{attribute addProperty BoxType "EK1100-0000-0018"}
{attribute addProperty Id "Beckhoff_EL34xxEK1122Beckhoff_EL34xxEK1122_54E02F3C162A_0001_EL3403_0000_0017EL3403_4661793D60275.25A_0002_EL3403_0000_0018EL3403_602DA43960275.25A_0003_EL3403_0000_0019EL3403_602DA43960275.25A_0004_EL3403_0000_0020EL3403_602DA43960275.25A_0005_EL3403_0000_0021EL3403_602DA43960275.25A_0006_EL3403_0000_0022EL3403_6F016EBB57071.25A_0007_EL3403_0000_0023EL3403_6F016EBB57071.25A_0008_EL3403_0010_0017EL3403_4661793D60275.25A_0009_EL3403_0010_0018EL3403_602DA43960275.25A_0010_EL3403_0010_0019EL3403_602DA43960275.25A_0011_EL3403_0010_0020EL3403_602DA43960275.25A_0012_EL3403_0010_0021EL3403_602DA43960275.25A_0013_EL3403_0010_0022EL3403_6F016EBB57071.25A_0014_EL3403_0010_0023EL3403_6F016EBB57071.25A_0015_EL3403_0010_0024EL3403_6F016EBB57071.25A_0016_EL3403_0026_0017EL3403_4661793D60275.25A_0017_EL3403_0026_0018EL3403_602DA43960275.25A_0018_EL3403_0026_0019EL3403_602DA43960275.25A_0019_EL3403_0026_0020EL3403_602DA43960275.25A_0020_EL3403_0026_0021EL3403_602DA43960275.25A_0021_EL3403_0026_0022EL3403_6F016EBB57071.25A_0022_EL3403_0026_0023EL3403_6F016EBB57071.25A_0023_EL3403_0026_0024EL3403_6F016EBB57071.25A_0024_EL3403_0100_0017EL3403_4661793D60275.25A_0025_EL3403_0100_0018EL3403_602DA43960275.25A_0026_EL3403_0100_0019EL3403_602DA43960275.25A_0027_EL3403_0100_0020EL3403_602DA43960275.25A_0028_EL3403_0100_0021EL3403_602DA43960275.25A_0029_EL3403_0100_0022EL3403_6F016EBB57071.25A_0030_EL3403_0100_0023EL3403_6F016EBB57071.25A_0031_EL3403_0100_0024EL3403_6F016EBB57071.25A_0032_EL3403_0111_0017EL3403_4661793D60275.25A_0033_EL3403_0111_0018EL3403_602DA43960275.25A_0034_EL3403_0111_0019EL3403_602DA43960275.25A_0035_EL3403_0111_0020EL3403_602DA43960275.25A_0036_EL3403_0111_0021EL3403_602DA43960275.25A_0037_EL3403_0111_0022EL3403_6F016EBB57071.25A_0038_EL3403_0111_0023EL3403_6F016EBB57071.25A_0039_EL3403_0111_0024EL3403_6F016EBB57071.25A_0040_EL3403_0126_0017EL3403_4661793D60275.25A_0041_EL3403_0126_0018EL3403_602DA43960275.25A_0042_EL3403_0126_0019EL3403_602DA43960275.25A_0043_EL3403_0126_0020EL3403_602DA43960275.25A_0044_EL3403_0126_0021EL3403_602DA43960275.25A_0045_EL3403_0126_0022EL3403_6F016EBB57071.25A_0046_EL3403_0126_0023EL3403_6F016EBB57071.25A_0047_EL3403_0126_0024EL3403_6F016EBB57071.25A_0048_EL3403_0333_0023EL3403_6F016EBB57071.25A_0049_EL3403_0333_0024EL3403_6F016EBB57071.25A_0050_EL3413_0000_0016EL3413_DFA511C864280.25A_0051_EL3413_0000_0017EL3413_DFA511C864280.25A_0052_EL3413_0000_0018EL3413_DFA511C864280.25A_0053_EL3413_0000_0019EL3413_BFE9962F64280.25A_0054_EL3413_0000_0020EL3413_BFE9962F64280.25A_0055_EL3413_0001_0016EL3413_BFE9962F64280.25A_0056_EL3413_0001_0017EL3413_BFE9962F64280.25A_0057_EL3413_0120_0017EL3413_DFA511C864280.25A_0058_EL3413_0001_0018EL3413_BFE9962F64280.25A_0059_EL3413_0120_0018EL3413_BFE9962F64280.25A_0060_EL3413_0120_0019EL3413_BFE9962F64280.25A_0061_EL3423_0000_0016EL3423_8712F12C1506188.25A_0062_EL3423_0000_0017EL3423_C8A9BC881506188.25A_0063_EL3423_0000_0018EL3423_C8A9BC881506188.25A_0064_EL3423_0000_0019EL3423_C8A9BC881506188.25A_0065_EL3423_0000_0020EL3423_AE18C60F930116.25A_0066_EL3423_0000_0021EL3423_AE18C60F930116.25A_0067_EL3433_0000_0016EL3433_BFE9962F64280.25A_0068_EL3433_0000_0017EL3433_BFE9962F64280.25A_0069_EL3433_0000_0018EL3433_BFE9962F64280.25A_0070_EL3443_0000_0016EL3443_2BD502B51650206.25A_0071_EL3443_0000_0017EL3443_538373741650206.25A_0072_EL3443_0000_0018EL3443_538373741650206.25A_0073_EL3443_0000_0019EL3443_538373741650206.25A_0074_EL3443_0000_0020EL3443_2BD502B51650206.25A_0075_EL3443_0000_0021EL3443_2BD502B51650206.25A_0076_EL3443_0010_0016EL3443_2BD502B51650206.25A_0077_EL3443_0010_0017EL3443_538373741650206.25A_0078_EL3443_0010_0018EL3443_538373741650206.25A_0079_EL3443_0010_0019EL3443_538373741650206.25A_0080_EL3443_0010_0020EL3443_2BD502B51650206.25A_0081_EL3443_0010_0021EL3443_2BD502B51650206.25A_0082_EL3443_0011_0018EL3443_538373741650206.25A_0083_EL3443_0011_0019EL3443_538373741650206.25A_0084_EL3443_0011_0020EL3443_2BD502B51650206.25A_0085_EL3443_0011_0021EL3443_2BD502B51650206.25A_0086_EL3443_0013_0018EL3443_538373741650206.25A_0087_EL3443_0013_0019EL3443_538373741650206.25A_0088_EL3443_0013_0020EL3443_2BD502B51650206.25A_0089_EL3443_0013_0021EL3443_2BD502B51650206.25A_0090_EL3446_0000_0016EL3446_80BBA9A057872.25A_0091_EL3446_0000_0017EL3446_80BBA9A057872.25A_0092_EL3453_0000_0017EL3453_10B71D421202150.25A_0093_EL3453_0000_0018EL3453_BDDFEB0B1194149.25A_0094_EL3453_0000_0019EL3453_BDDFEB0B1194149.25A_0095_EL3453_0000_0020EL3453_10B71D421202150.25A_0096_EL3453_0000_0021EL3453_10B71D421202150.25A_0097_EL3453_0100_0021EL3453_10B71D421202150.25A_0098_EL3483_0000_0016EL3483_4A23656431439.25A_0099_EL3483_0000_0017EL3483_4A23656431439.25A_0100_EL3483_0000_0018EL3483_4A23656431439.25A_0101_EL3483_0000_0019EL3483_4A23656431439.25A_0102_EL3483_0000_0020EL3483_4A23656431439.25A_0103_EL3483_0000_0021EL3483_4A23656431439.25A_0104_EL3483_0060_0018EL3483_2724D36850663.25A_0105_EL3483_0060_0019EL3483_2724D36850663.25A_0106_EL3483_0060_0020EL3483_EF2C452150663.25A_0107_EL3483_0060_0021EL3483_EF2C452150663.25"}
{attribute addProperty CRC "1278133200"}
{attribute addProperty SizeInBites "91038"}
{attribute addProperty SizeInBytes "11379.75"}
TYPE Beckhoff_EL34xx_4C2EC3D0 EXTENDS EK1100_179A0949 :
STRUCT
	{attribute addProperty Name "Beckhoff_EL34xxEK1122"}
	Beckhoff_EL34xxEK1122 : Beckhoff_EL34xxEK1122_54E02F3C;
	{attribute addProperty Name "A_0001_EL3403_0000_0017"}
	A_0001_EL3403_0000_0017 : EL3403_4661793D;
	{attribute addProperty Name "A_0002_EL3403_0000_0018"}
	A_0002_EL3403_0000_0018 : EL3403_602DA439;
	{attribute addProperty Name "A_0003_EL3403_0000_0019"}
	A_0003_EL3403_0000_0019 : EL3403_602DA439;
	{attribute addProperty Name "A_0004_EL3403_0000_0020"}
	A_0004_EL3403_0000_0020 : EL3403_602DA439;
	{attribute addProperty Name "A_0005_EL3403_0000_0021"}
	A_0005_EL3403_0000_0021 : EL3403_602DA439;
	{attribute addProperty Name "A_0006_EL3403_0000_0022"}
	A_0006_EL3403_0000_0022 : EL3403_6F016EBB;
	{attribute addProperty Name "A_0007_EL3403_0000_0023"}
	A_0007_EL3403_0000_0023 : EL3403_6F016EBB;
	{attribute addProperty Name "A_0008_EL3403_0010_0017"}
	A_0008_EL3403_0010_0017 : EL3403_4661793D;
	{attribute addProperty Name "A_0009_EL3403_0010_0018"}
	A_0009_EL3403_0010_0018 : EL3403_602DA439;
	{attribute addProperty Name "A_0010_EL3403_0010_0019"}
	A_0010_EL3403_0010_0019 : EL3403_602DA439;
	{attribute addProperty Name "A_0011_EL3403_0010_0020"}
	A_0011_EL3403_0010_0020 : EL3403_602DA439;
	{attribute addProperty Name "A_0012_EL3403_0010_0021"}
	A_0012_EL3403_0010_0021 : EL3403_602DA439;
	{attribute addProperty Name "A_0013_EL3403_0010_0022"}
	A_0013_EL3403_0010_0022 : EL3403_6F016EBB;
	{attribute addProperty Name "A_0014_EL3403_0010_0023"}
	A_0014_EL3403_0010_0023 : EL3403_6F016EBB;
	{attribute addProperty Name "A_0015_EL3403_0010_0024"}
	A_0015_EL3403_0010_0024 : EL3403_6F016EBB;
	{attribute addProperty Name "A_0016_EL3403_0026_0017"}
	A_0016_EL3403_0026_0017 : EL3403_4661793D;
	{attribute addProperty Name "A_0017_EL3403_0026_0018"}
	A_0017_EL3403_0026_0018 : EL3403_602DA439;
	{attribute addProperty Name "A_0018_EL3403_0026_0019"}
	A_0018_EL3403_0026_0019 : EL3403_602DA439;
	{attribute addProperty Name "A_0019_EL3403_0026_0020"}
	A_0019_EL3403_0026_0020 : EL3403_602DA439;
	{attribute addProperty Name "A_0020_EL3403_0026_0021"}
	A_0020_EL3403_0026_0021 : EL3403_602DA439;
	{attribute addProperty Name "A_0021_EL3403_0026_0022"}
	A_0021_EL3403_0026_0022 : EL3403_6F016EBB;
	{attribute addProperty Name "A_0022_EL3403_0026_0023"}
	A_0022_EL3403_0026_0023 : EL3403_6F016EBB;
	{attribute addProperty Name "A_0023_EL3403_0026_0024"}
	A_0023_EL3403_0026_0024 : EL3403_6F016EBB;
	{attribute addProperty Name "A_0024_EL3403_0100_0017"}
	A_0024_EL3403_0100_0017 : EL3403_4661793D;
	{attribute addProperty Name "A_0025_EL3403_0100_0018"}
	A_0025_EL3403_0100_0018 : EL3403_602DA439;
	{attribute addProperty Name "A_0026_EL3403_0100_0019"}
	A_0026_EL3403_0100_0019 : EL3403_602DA439;
	{attribute addProperty Name "A_0027_EL3403_0100_0020"}
	A_0027_EL3403_0100_0020 : EL3403_602DA439;
	{attribute addProperty Name "A_0028_EL3403_0100_0021"}
	A_0028_EL3403_0100_0021 : EL3403_602DA439;
	{attribute addProperty Name "A_0029_EL3403_0100_0022"}
	A_0029_EL3403_0100_0022 : EL3403_6F016EBB;
	{attribute addProperty Name "A_0030_EL3403_0100_0023"}
	A_0030_EL3403_0100_0023 : EL3403_6F016EBB;
	{attribute addProperty Name "A_0031_EL3403_0100_0024"}
	A_0031_EL3403_0100_0024 : EL3403_6F016EBB;
	{attribute addProperty Name "A_0032_EL3403_0111_0017"}
	A_0032_EL3403_0111_0017 : EL3403_4661793D;
	{attribute addProperty Name "A_0033_EL3403_0111_0018"}
	A_0033_EL3403_0111_0018 : EL3403_602DA439;
	{attribute addProperty Name "A_0034_EL3403_0111_0019"}
	A_0034_EL3403_0111_0019 : EL3403_602DA439;
	{attribute addProperty Name "A_0035_EL3403_0111_0020"}
	A_0035_EL3403_0111_0020 : EL3403_602DA439;
	{attribute addProperty Name "A_0036_EL3403_0111_0021"}
	A_0036_EL3403_0111_0021 : EL3403_602DA439;
	{attribute addProperty Name "A_0037_EL3403_0111_0022"}
	A_0037_EL3403_0111_0022 : EL3403_6F016EBB;
	{attribute addProperty Name "A_0038_EL3403_0111_0023"}
	A_0038_EL3403_0111_0023 : EL3403_6F016EBB;
	{attribute addProperty Name "A_0039_EL3403_0111_0024"}
	A_0039_EL3403_0111_0024 : EL3403_6F016EBB;
	{attribute addProperty Name "A_0040_EL3403_0126_0017"}
	A_0040_EL3403_0126_0017 : EL3403_4661793D;
	{attribute addProperty Name "A_0041_EL3403_0126_0018"}
	A_0041_EL3403_0126_0018 : EL3403_602DA439;
	{attribute addProperty Name "A_0042_EL3403_0126_0019"}
	A_0042_EL3403_0126_0019 : EL3403_602DA439;
	{attribute addProperty Name "A_0043_EL3403_0126_0020"}
	A_0043_EL3403_0126_0020 : EL3403_602DA439;
	{attribute addProperty Name "A_0044_EL3403_0126_0021"}
	A_0044_EL3403_0126_0021 : EL3403_602DA439;
	{attribute addProperty Name "A_0045_EL3403_0126_0022"}
	A_0045_EL3403_0126_0022 : EL3403_6F016EBB;
	{attribute addProperty Name "A_0046_EL3403_0126_0023"}
	A_0046_EL3403_0126_0023 : EL3403_6F016EBB;
	{attribute addProperty Name "A_0047_EL3403_0126_0024"}
	A_0047_EL3403_0126_0024 : EL3403_6F016EBB;
	{attribute addProperty Name "A_0048_EL3403_0333_0023"}
	A_0048_EL3403_0333_0023 : EL3403_6F016EBB;
	{attribute addProperty Name "A_0049_EL3403_0333_0024"}
	A_0049_EL3403_0333_0024 : EL3403_6F016EBB;
	{attribute addProperty Name "A_0050_EL3413_0000_0016"}
	A_0050_EL3413_0000_0016 : EL3413_DFA511C8;
	{attribute addProperty Name "A_0051_EL3413_0000_0017"}
	A_0051_EL3413_0000_0017 : EL3413_DFA511C8;
	{attribute addProperty Name "A_0052_EL3413_0000_0018"}
	A_0052_EL3413_0000_0018 : EL3413_DFA511C8;
	{attribute addProperty Name "A_0053_EL3413_0000_0019"}
	A_0053_EL3413_0000_0019 : EL3413_BFE9962F;
	{attribute addProperty Name "A_0054_EL3413_0000_0020"}
	A_0054_EL3413_0000_0020 : EL3413_BFE9962F;
	{attribute addProperty Name "A_0055_EL3413_0001_0016"}
	A_0055_EL3413_0001_0016 : EL3413_BFE9962F;
	{attribute addProperty Name "A_0056_EL3413_0001_0017"}
	A_0056_EL3413_0001_0017 : EL3413_BFE9962F;
	{attribute addProperty Name "A_0057_EL3413_0120_0017"}
	A_0057_EL3413_0120_0017 : EL3413_DFA511C8;
	{attribute addProperty Name "A_0058_EL3413_0001_0018"}
	A_0058_EL3413_0001_0018 : EL3413_BFE9962F;
	{attribute addProperty Name "A_0059_EL3413_0120_0018"}
	A_0059_EL3413_0120_0018 : EL3413_BFE9962F;
	{attribute addProperty Name "A_0060_EL3413_0120_0019"}
	A_0060_EL3413_0120_0019 : EL3413_BFE9962F;
	{attribute addProperty Name "A_0061_EL3423_0000_0016"}
	A_0061_EL3423_0000_0016 : EL3423_8712F12C;
	{attribute addProperty Name "A_0062_EL3423_0000_0017"}
	A_0062_EL3423_0000_0017 : EL3423_C8A9BC88;
	{attribute addProperty Name "A_0063_EL3423_0000_0018"}
	A_0063_EL3423_0000_0018 : EL3423_C8A9BC88;
	{attribute addProperty Name "A_0064_EL3423_0000_0019"}
	A_0064_EL3423_0000_0019 : EL3423_C8A9BC88;
	{attribute addProperty Name "A_0065_EL3423_0000_0020"}
	A_0065_EL3423_0000_0020 : EL3423_AE18C60F;
	{attribute addProperty Name "A_0066_EL3423_0000_0021"}
	A_0066_EL3423_0000_0021 : EL3423_AE18C60F;
	{attribute addProperty Name "A_0067_EL3433_0000_0016"}
	A_0067_EL3433_0000_0016 : EL3433_BFE9962F;
	{attribute addProperty Name "A_0068_EL3433_0000_0017"}
	A_0068_EL3433_0000_0017 : EL3433_BFE9962F;
	{attribute addProperty Name "A_0069_EL3433_0000_0018"}
	A_0069_EL3433_0000_0018 : EL3433_BFE9962F;
	{attribute addProperty Name "A_0070_EL3443_0000_0016"}
	A_0070_EL3443_0000_0016 : EL3443_2BD502B5;
	{attribute addProperty Name "A_0071_EL3443_0000_0017"}
	A_0071_EL3443_0000_0017 : EL3443_53837374;
	{attribute addProperty Name "A_0072_EL3443_0000_0018"}
	A_0072_EL3443_0000_0018 : EL3443_53837374;
	{attribute addProperty Name "A_0073_EL3443_0000_0019"}
	A_0073_EL3443_0000_0019 : EL3443_53837374;
	{attribute addProperty Name "A_0074_EL3443_0000_0020"}
	A_0074_EL3443_0000_0020 : EL3443_2BD502B5;
	{attribute addProperty Name "A_0075_EL3443_0000_0021"}
	A_0075_EL3443_0000_0021 : EL3443_2BD502B5;
	{attribute addProperty Name "A_0076_EL3443_0010_0016"}
	A_0076_EL3443_0010_0016 : EL3443_2BD502B5;
	{attribute addProperty Name "A_0077_EL3443_0010_0017"}
	A_0077_EL3443_0010_0017 : EL3443_53837374;
	{attribute addProperty Name "A_0078_EL3443_0010_0018"}
	A_0078_EL3443_0010_0018 : EL3443_53837374;
	{attribute addProperty Name "A_0079_EL3443_0010_0019"}
	A_0079_EL3443_0010_0019 : EL3443_53837374;
	{attribute addProperty Name "A_0080_EL3443_0010_0020"}
	A_0080_EL3443_0010_0020 : EL3443_2BD502B5;
	{attribute addProperty Name "A_0081_EL3443_0010_0021"}
	A_0081_EL3443_0010_0021 : EL3443_2BD502B5;
	{attribute addProperty Name "A_0082_EL3443_0011_0018"}
	A_0082_EL3443_0011_0018 : EL3443_53837374;
	{attribute addProperty Name "A_0083_EL3443_0011_0019"}
	A_0083_EL3443_0011_0019 : EL3443_53837374;
	{attribute addProperty Name "A_0084_EL3443_0011_0020"}
	A_0084_EL3443_0011_0020 : EL3443_2BD502B5;
	{attribute addProperty Name "A_0085_EL3443_0011_0021"}
	A_0085_EL3443_0011_0021 : EL3443_2BD502B5;
	{attribute addProperty Name "A_0086_EL3443_0013_0018"}
	A_0086_EL3443_0013_0018 : EL3443_53837374;
	{attribute addProperty Name "A_0087_EL3443_0013_0019"}
	A_0087_EL3443_0013_0019 : EL3443_53837374;
	{attribute addProperty Name "A_0088_EL3443_0013_0020"}
	A_0088_EL3443_0013_0020 : EL3443_2BD502B5;
	{attribute addProperty Name "A_0089_EL3443_0013_0021"}
	A_0089_EL3443_0013_0021 : EL3443_2BD502B5;
	{attribute addProperty Name "A_0090_EL3446_0000_0016"}
	A_0090_EL3446_0000_0016 : EL3446_80BBA9A0;
	{attribute addProperty Name "A_0091_EL3446_0000_0017"}
	A_0091_EL3446_0000_0017 : EL3446_80BBA9A0;
	{attribute addProperty Name "A_0092_EL3453_0000_0017"}
	A_0092_EL3453_0000_0017 : EL3453_10B71D42;
	{attribute addProperty Name "A_0093_EL3453_0000_0018"}
	A_0093_EL3453_0000_0018 : EL3453_BDDFEB0B;
	{attribute addProperty Name "A_0094_EL3453_0000_0019"}
	A_0094_EL3453_0000_0019 : EL3453_BDDFEB0B;
	{attribute addProperty Name "A_0095_EL3453_0000_0020"}
	A_0095_EL3453_0000_0020 : EL3453_10B71D42;
	{attribute addProperty Name "A_0096_EL3453_0000_0021"}
	A_0096_EL3453_0000_0021 : EL3453_10B71D42;
	{attribute addProperty Name "A_0097_EL3453_0100_0021"}
	A_0097_EL3453_0100_0021 : EL3453_10B71D42;
	{attribute addProperty Name "A_0098_EL3483_0000_0016"}
	A_0098_EL3483_0000_0016 : EL3483_4A236564;
	{attribute addProperty Name "A_0099_EL3483_0000_0017"}
	A_0099_EL3483_0000_0017 : EL3483_4A236564;
	{attribute addProperty Name "A_0100_EL3483_0000_0018"}
	A_0100_EL3483_0000_0018 : EL3483_4A236564;
	{attribute addProperty Name "A_0101_EL3483_0000_0019"}
	A_0101_EL3483_0000_0019 : EL3483_4A236564;
	{attribute addProperty Name "A_0102_EL3483_0000_0020"}
	A_0102_EL3483_0000_0020 : EL3483_4A236564;
	{attribute addProperty Name "A_0103_EL3483_0000_0021"}
	A_0103_EL3483_0000_0021 : EL3483_4A236564;
	{attribute addProperty Name "A_0104_EL3483_0060_0018"}
	A_0104_EL3483_0060_0018 : EL3483_2724D368;
	{attribute addProperty Name "A_0105_EL3483_0060_0019"}
	A_0105_EL3483_0060_0019 : EL3483_2724D368;
	{attribute addProperty Name "A_0106_EL3483_0060_0020"}
	A_0106_EL3483_0060_0020 : EL3483_EF2C4521;
	{attribute addProperty Name "A_0107_EL3483_0060_0021"}
	A_0107_EL3483_0060_0021 : EL3483_EF2C4521;
END_STRUCT
END_TYPE

(* stored: Version 1.2.0.0, ProductVersion 3.1.4024.9
   DUT Beckhoff_EL34xx_4C2EC3D0: Id {2bf12485-8214-41c2-a7b1-48c152b9b8e6} *)
